// TIA Portal project "OpennessTest" (V17)

(* hardware
DEVICE "S7-1200 station_1"  S7-1200 Station
   slot 0: "Rack_0"  S7-1200 Rack  Rack  V1.0
   slot 1: "PLC_Valdymas"  CPU 1214C DC/DC/Rly  6ES7 214-1HG40-0XB0  V4.5
*)

// ===== PLC "PLC_Valdymas"  CPU 1214C DC/DC/Rly =====

FUNCTION_BLOCK "DivideFB"   // FB1, SCL
{ S7_Optimized_Access := 'TRUE' }
VERSION : 0.1
   VAR_INPUT
      in0 : Real;
      in1 : Real;
   END_VAR
   VAR_OUTPUT
      res : Real;
   END_VAR
BEGIN
   #res := #in0 / #in1;
END_FUNCTION_BLOCK

FUNCTION_BLOCK "MultipleFB"   // FB2, SCL
{ S7_Optimized_Access := 'TRUE' }
VERSION : 0.1
   VAR_INPUT
      in0 : Int;
      in1 : Int;
   END_VAR
   VAR_OUTPUT
      res : Int;
   END_VAR
BEGIN
   #res := #in0 * #in1;
END_FUNCTION_BLOCK

FUNCTION_BLOCK "SubstractFB"   // FB3, SCL
{ S7_Optimized_Access := 'TRUE' }
VERSION : 0.1
   VAR_INPUT
      in0 : Int;
      in1 : Int;
   END_VAR
   VAR_OUTPUT
      res : Int;
   END_VAR
BEGIN
   #res := #in0 - #in1;
END_FUNCTION_BLOCK

FUNCTION_BLOCK "SumFB"   // FB4, SCL
{ S7_Optimized_Access := 'TRUE' }
VERSION : 0.1
   VAR_INPUT
      in0 : Int;
      in1 : Int;
   END_VAR
   VAR_OUTPUT
      res : Int;
   END_VAR
BEGIN
   #res := #in0 + #in1;
END_FUNCTION_BLOCK

ORGANIZATION_BLOCK "Main"   // OB1, LAD, ProgramCycle
TITLE = "Main Program Sweep (Cycle)"
{ S7_Optimized_Access := 'TRUE' }
VERSION : 0.1
   VAR_INPUT
      Initial_Call : Bool;   // Initial call of this OB
      Remanence : Bool;   // =True, if remanent data are available
   END_VAR
BEGIN
END_ORGANIZATION_BLOCK